TYPE EtcMasterBase_62654B43 :
STRUCT
END_STRUCT
END_TYPE

(* stored: Version 1.2.0.0, ProductVersion 3.1.4024.9
   DUT EtcMasterBase_62654B43: Id {cade258b-7e39-4fad-b66c-626abfcd7b72} *)
